Staubli VAL3: alreadyExist.pgx

program alreadyExist(string& x_sName[], bool& x_bUndo[])
  local num l_nX
  local num l_nY
  local string l_sString
begin
  // look if the trajectory already exist
  l_nX=40-use:nBottomX-1
  l_nY=use:nBottomY+1
  call language:message(l_sString,21)
  call use:type(l_nX,l_nY,l_sString)
  // read the new trajectory
  call use:read(l_nX+len(l_sString),l_nY,x_sName,10,false)
  if !use:bUseEscape
    call set:find(x_sName,x_bUndo)
    if x_bUndo
      call language:message(x_sName,-2)
      popUpMsg(x_sName)
    endIf
  else
    x_bUndo=true
  endIf
end
